FUNCTION_BLOCK LeadingCar
  (* Standard: 61499-2 *)
  (* Version 0.1, 2015-00-08, SYY, SYY-PC *)
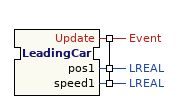
  EVENT_OUTPUT
    Update WITH pos1, speed1;
  END_EVENT
  VAR_OUTPUT
    pos1 : LREAL := 100;
    speed1 : LREAL := 1;
  END_VAR
  VAR
    v : REAL;
    x : LREAL;
    d : LREAL;
    k : INT;
    t : INT := 0;
    random_t : INT;
  END_VAR
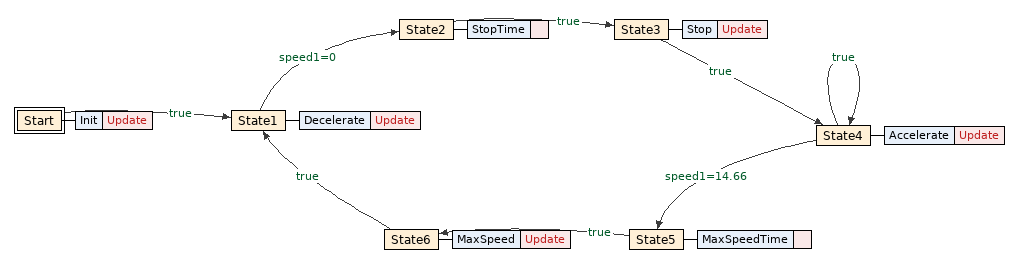
  EC_STATES
    Start : Init -> Update;
    State1 : Decelerate -> Update;
    State3 : Stop -> Update;
    State4 : Accelerate -> Update;
    State6 : MaxSpeed -> Update;
    State2 : StopTime;
    State5 : MaxSpeedTime;
  END_STATES
  EC_TRANSITIONS
    Start TO State1 := true;
    State1 TO State2 := speed1=0;
    State3 TO State4 := true;
    State4 TO State5 := speed1=14.66;
    State4 TO State4 := true;
    State6 TO State1 := true;
    State2 TO State3 := true;
    State5 TO State6 := true;
  END_TRANSITIONS
  ALGORITHM Init IN C:
me->d = 0.01;
me->speed1 = 1;
me->pos1 = 32.5;
me->k = 37;
  END_ALGORITHM
  ALGORITHM Decelerate IN C:
me->v = me->speed1;
me->x = me->pos1;
//me->speed1 = -0.0097*me->k*me->k - 0.0105*me->k + 14.707;
me->speed1 = 0;
//me->pos1 = me->x + me->d * me->v;
me->pos1 = me->pos1 + 3.81;
me->k = me->k + 1;

if(me->speed1<=0){
  me->speed1 = 0;
  me->k = 0;
  me->t = 0;
}

printf("Leading car decelerates (Position: %3.8f, Speed: %3.8f)\n", me->pos1, me->speed1);
  END_ALGORITHM
  ALGORITHM Accelerate IN C:
me->v = me->speed1;
me->x = me->pos1;
me->k = me->k + 1;
//me->speed1 = 0.0097*me->k*me->k + 0.0112*me->k - 0.0482;
me->speed1 = 14.66;
//me->pos1 = me->x + me->d * me->v;
me->pos1 = me->pos1 + 2.05;

if(me->speed1>=14.66){
  me->speed1 = 14.66;
  me->k = 0;
  me->t = 0;
}

printf("Leading car accelerates (Position: %3.8f, Speed: %3.8f)\n", me->pos1, me->speed1);
  END_ALGORITHM
  ALGORITHM MaxSpeed IN C:
me->x = me->pos1;
me->v = me->speed1;
me->k = me->k + 1;
//me->pos1 = me->x + me->d * me->v;
me->pos1 = me->pos1 + 29.18;
printf("Leading car (Position: %3.8f, Speed: %3.8f)\n", me->pos1, me->speed1);

if(me->k*me->d==me->random_t){
  me->k = 1;
  me->t = me->random_t;
}
  END_ALGORITHM
  ALGORITHM Stop IN C:
me->x = me->pos1;
me->v = me->speed1;
me->k = me->k + 1;
//me->pos1 = me->x + me->d * me->v;
printf("Leading car (Position: %3.8f, Speed: %3.8f)\n", me->pos1, me->speed1);

if(me->k*me->d==me->random_t){
  me->k = 1;
  me->t = me->random_t;
}
  END_ALGORITHM
  ALGORITHM StopTime IN C:
//srand(time(NULL));
//int temp=rand()%2;
//if (temp==1){
//me->random_t=9;
//}else if(temp==0){
//me->random_t=6;
//}
me->random_t=6;
  END_ALGORITHM
  ALGORITHM MaxSpeedTime IN C:
//srand(time(NULL));
//int temp=rand()%2;
//if (temp==1){
//me->random_t=1;
//}else if(temp==0){
//me->random_t=3;
//}
me->random_t=2;
  END_ALGORITHM
END_FUNCTION_BLOCK
